// TIA Portal V16 export
// export: Created 2021-07-22T09:12:31.8066406Z, ExportSetting WithDefaults, WithReadOnly, DisplayName Totally Integrated Automation Portal, DisplayVersion V16 Update 3, DisplayName TIA Portal Version Control Interface, DisplayVersion V16 Update 2, DisplayName TIA Portal Openness, DisplayVersion V16 Update 3, DisplayName SINAMICS Startdrive Advanced, DisplayVersion V16, DisplayName SINAMICS Startdrive G130, G150, S120, S150, SINAMICS MV, S210, DisplayVersion V16, DisplayName SINAMICS Startdrive G110M, G120, G120C, G120D, G120P, DisplayVersion V16, DisplayName STEP 7 Professional, DisplayVersion V16 Update 3, DisplayName SIMATIC Energy Suite, DisplayVersion V16, DisplayName STEP 7 Safety, DisplayVersion V16, DisplayName WinCC Advanced, DisplayVersion V16 Update 3
Screen "Terziario"  1366x768, Number=4, Template=Intestazione
  ScreenLayer 
    TextField "Casella di testo_1" at 608,60 size 151x38  Text="CABINA 3"
    Button "Pulsante_2" at 1300,689 size 59x32  Mode=Text, TextOff="Next", TextOn="Text"
      on Click: ActivateScreen(Screen name := pagina_successiva, Object number := 0)
    Button "Pulsante_3" at 1236,690 size 59x32  Mode=Text, TextOff="Prev.", TextOn="Text"
      on Click: ActivateScreen(Screen name := pagina_precedente, Object number := 0)
    Button "Pulsante_4" at 1300,725 size 59x32  Mode=Text, TextOff="Home", TextOn="Text"
      on Click: ActivateScreen(Screen name := home, Object number := 0)
